// TIA Portal V17 export
// export: Created 2025-03-12T15:33:06.1888493Z, ExportSetting WithDefaults, DisplayName Totally Integrated Automation Portal, DisplayVersion V17 Update 8, DisplayName TIA Portal Openness, DisplayVersion V17 Update 8, DisplayName TIA Portal Version Control Interface, DisplayVersion V17, DisplayName SINAMICS Startdrive Advanced, DisplayVersion V17 SP2, DisplayName SINAMICS Startdrive G110M, G120, G120C, G120D, G120P, G115D, DisplayVersion V17 SP2, DisplayName SINAMICS Startdrive G130, G150, S120, S150, SINAMICS MV, S210, DisplayVersion V17 SP2, DisplayName STEP 7 Professional, DisplayVersion V17 Update 8, DisplayName SINUMERIK ONE STEP 7 Toolbox, DisplayVersion V17 Update 12, DisplayName SINUMERIK 840D sl STEP 7 Toolbox, DisplayVersion V17 Update 12, DisplayName STEP 7 Safety, DisplayVersion V17 Update 6, DisplayName WinCC Advanced, DisplayVersion V17 Update 8
FUNCTION_BLOCK "Main_Safety_RTG1"   // FB1010, F_LAD
{ S7_Optimized_Access := 'TRUE' }
VERSION : 0.1
// stored: AutoNumber false, IsIECCheckEnabled false, UDAEnableTagReadback false
   VAR
      ACK_GL_Instance : ACK_GL;
   END_VAR
BEGIN

REGION Network 1: RECEIVE SAFE I/O FROM KF900
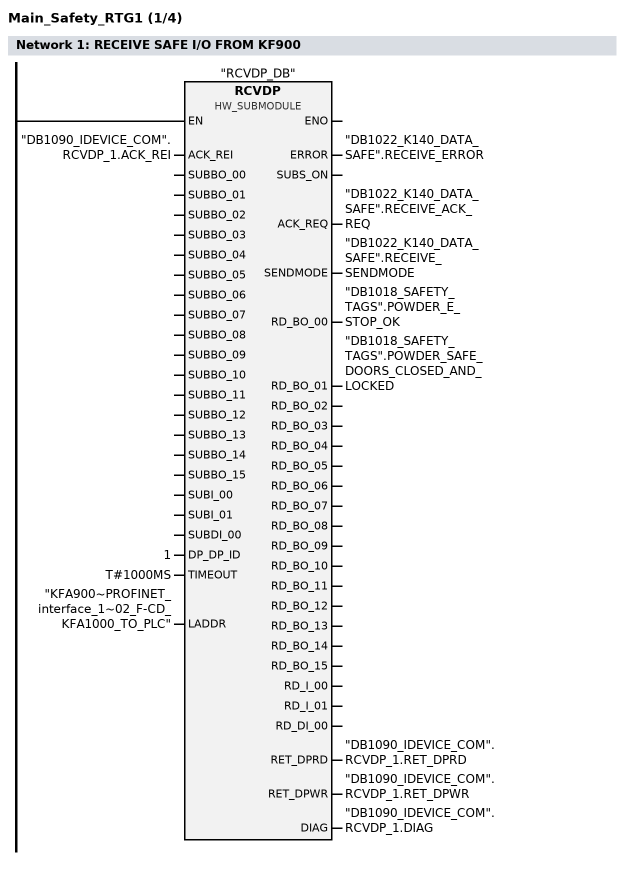
   RUNG wire#powerrail
      { S7_Templates := "laddr_type := HW_SUBMODULE" } "RCVDP_DB".RCVDP(ACK_REI := "DB1090_IDEVICE_COM".RCVDP_1.ACK_REI, SUBBO_00 :=, SUBBO_01 :=, SUBBO_02 :=, SUBBO_03 :=, SUBBO_04 :=, SUBBO_05 :=, SUBBO_06 :=, SUBBO_07 :=, SUBBO_08 :=, SUBBO_09 :=, SUBBO_10 :=, SUBBO_11 :=, SUBBO_12 :=, SUBBO_13 :=, SUBBO_14 :=, SUBBO_15 :=, SUBI_00 :=, SUBI_01 :=, SUBDI_00 :=, DP_DP_ID := 1, TIMEOUT := T#1000MS, LADDR := "KFA900~PROFINET_interface_1~02_F-CD_KFA1000_TO_PLC", ERROR => "DB1022_K140_DATA_SAFE".RECEIVE_ERROR, SUBS_ON =>, ACK_REQ => "DB1022_K140_DATA_SAFE".RECEIVE_ACK_REQ, SENDMODE => "DB1022_K140_DATA_SAFE".RECEIVE_SENDMODE, RD_BO_00 => "DB1018_SAFETY_TAGS".POWDER_E_STOP_OK, RD_BO_01 => "DB1018_SAFETY_TAGS".POWDER_SAFE_DOORS_CLOSED_AND_LOCKED, RD_BO_02 =>, RD_BO_03 =>, RD_BO_04 =>, RD_BO_05 =>, RD_BO_06 =>, RD_BO_07 =>, RD_BO_08 =>, RD_BO_09 =>, RD_BO_10 =>, RD_BO_11 =>, RD_BO_12 =>, RD_BO_13 =>, RD_BO_14 =>, RD_BO_15 =>, RD_I_00 =>, RD_I_01 =>, RD_DI_00 =>, RET_DPRD => "DB1090_IDEVICE_COM".RCVDP_1.RET_DPRD, RET_DPWR => "DB1090_IDEVICE_COM".RCVDP_1.RET_DPWR, DIAG => "DB1090_IDEVICE_COM".RCVDP_1.DIAG)
   END_RUNG
   // the same network as SCL:
   "RCVDP_DB"(ACK_REI := "DB1090_IDEVICE_COM".RCVDP_1.ACK_REI,   // RCVDP
              DP_DP_ID := 1,
              TIMEOUT := T#1000MS,
              LADDR := "KFA900~PROFINET_interface_1~02_F-CD_KFA1000_TO_PLC",
              ERROR => "DB1022_K140_DATA_SAFE".RECEIVE_ERROR,
              ACK_REQ => "DB1022_K140_DATA_SAFE".RECEIVE_ACK_REQ,
              SENDMODE => "DB1022_K140_DATA_SAFE".RECEIVE_SENDMODE,
              RD_BO_00 => "DB1018_SAFETY_TAGS".POWDER_E_STOP_OK,
              RD_BO_01 => "DB1018_SAFETY_TAGS".POWDER_SAFE_DOORS_CLOSED_AND_LOCKED,
              RET_DPRD => "DB1090_IDEVICE_COM".RCVDP_1.RET_DPRD,
              RET_DPWR => "DB1090_IDEVICE_COM".RCVDP_1.RET_DPWR,
              DIAG => "DB1090_IDEVICE_COM".RCVDP_1.DIAG);
END_REGION

REGION Network 2: RECEIVE SAFE I/O FROM ETXETAR CELL
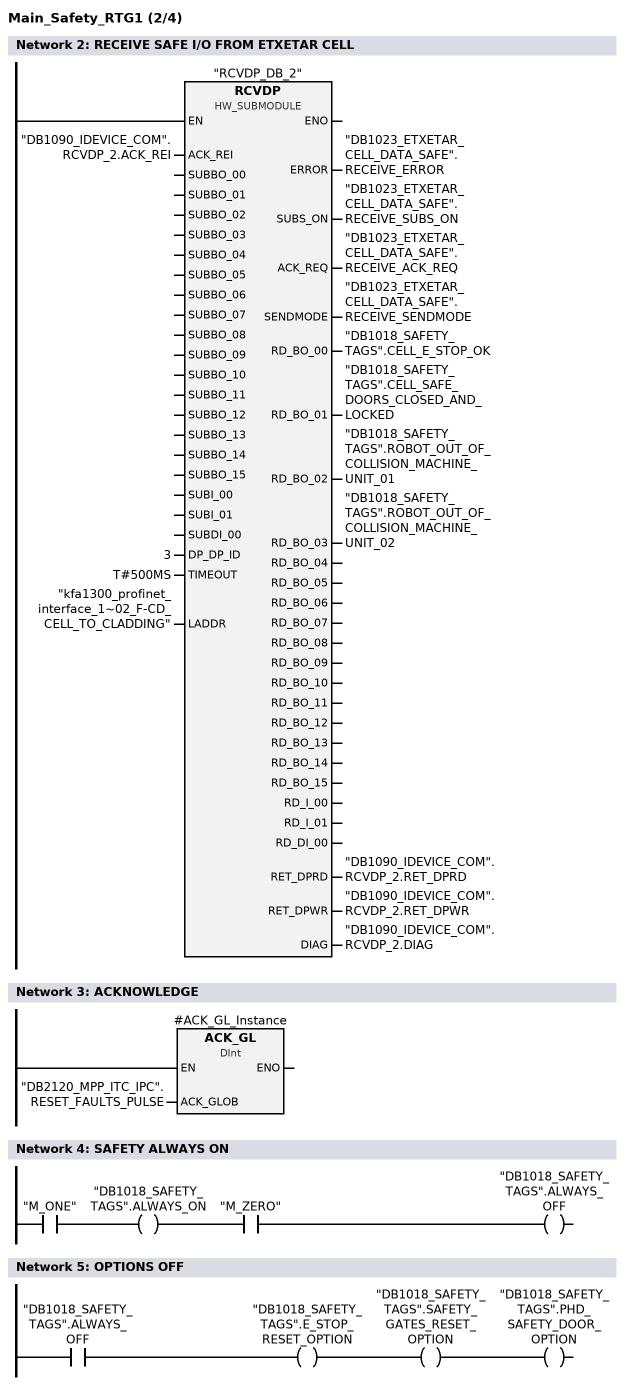
   RUNG wire#powerrail
      { S7_Templates := "laddr_type := HW_SUBMODULE" } "RCVDP_DB_2".RCVDP(ACK_REI := "DB1090_IDEVICE_COM".RCVDP_2.ACK_REI, SUBBO_00 :=, SUBBO_01 :=, SUBBO_02 :=, SUBBO_03 :=, SUBBO_04 :=, SUBBO_05 :=, SUBBO_06 :=, SUBBO_07 :=, SUBBO_08 :=, SUBBO_09 :=, SUBBO_10 :=, SUBBO_11 :=, SUBBO_12 :=, SUBBO_13 :=, SUBBO_14 :=, SUBBO_15 :=, SUBI_00 :=, SUBI_01 :=, SUBDI_00 :=, DP_DP_ID := 3, TIMEOUT := T#500MS, LADDR := "kfa1300_profinet_interface_1~02_F-CD_CELL_TO_CLADDING", ERROR => "DB1023_ETXETAR_CELL_DATA_SAFE".RECEIVE_ERROR, SUBS_ON => "DB1023_ETXETAR_CELL_DATA_SAFE".RECEIVE_SUBS_ON, ACK_REQ => "DB1023_ETXETAR_CELL_DATA_SAFE".RECEIVE_ACK_REQ, SENDMODE => "DB1023_ETXETAR_CELL_DATA_SAFE".RECEIVE_SENDMODE, RD_BO_00 => "DB1018_SAFETY_TAGS".CELL_E_STOP_OK, RD_BO_01 => "DB1018_SAFETY_TAGS".CELL_SAFE_DOORS_CLOSED_AND_LOCKED, RD_BO_02 => "DB1018_SAFETY_TAGS".ROBOT_OUT_OF_COLLISION_MACHINE_UNIT_01, RD_BO_03 => "DB1018_SAFETY_TAGS".ROBOT_OUT_OF_COLLISION_MACHINE_UNIT_02, RD_BO_04 =>, RD_BO_05 =>, RD_BO_06 =>, RD_BO_07 =>, RD_BO_08 =>, RD_BO_09 =>, RD_BO_10 =>, RD_BO_11 =>, RD_BO_12 =>, RD_BO_13 =>, RD_BO_14 =>, RD_BO_15 =>, RD_I_00 =>, RD_I_01 =>, RD_DI_00 =>, RET_DPRD => "DB1090_IDEVICE_COM".RCVDP_2.RET_DPRD, RET_DPWR => "DB1090_IDEVICE_COM".RCVDP_2.RET_DPWR, DIAG => "DB1090_IDEVICE_COM".RCVDP_2.DIAG)
   END_RUNG
   // the same network as SCL:
   "RCVDP_DB_2"(ACK_REI := "DB1090_IDEVICE_COM".RCVDP_2.ACK_REI,   // RCVDP
                DP_DP_ID := 3,
                TIMEOUT := T#500MS,
                LADDR := "kfa1300_profinet_interface_1~02_F-CD_CELL_TO_CLADDING",
                ERROR => "DB1023_ETXETAR_CELL_DATA_SAFE".RECEIVE_ERROR,
                SUBS_ON => "DB1023_ETXETAR_CELL_DATA_SAFE".RECEIVE_SUBS_ON,
                ACK_REQ => "DB1023_ETXETAR_CELL_DATA_SAFE".RECEIVE_ACK_REQ,
                SENDMODE => "DB1023_ETXETAR_CELL_DATA_SAFE".RECEIVE_SENDMODE,
                RD_BO_00 => "DB1018_SAFETY_TAGS".CELL_E_STOP_OK,
                RD_BO_01 => "DB1018_SAFETY_TAGS".CELL_SAFE_DOORS_CLOSED_AND_LOCKED,
                RD_BO_02 => "DB1018_SAFETY_TAGS".ROBOT_OUT_OF_COLLISION_MACHINE_UNIT_01,
                RD_BO_03 => "DB1018_SAFETY_TAGS".ROBOT_OUT_OF_COLLISION_MACHINE_UNIT_02,
                RET_DPRD => "DB1090_IDEVICE_COM".RCVDP_2.RET_DPRD,
                RET_DPWR => "DB1090_IDEVICE_COM".RCVDP_2.RET_DPWR,
                DIAG => "DB1090_IDEVICE_COM".RCVDP_2.DIAG);
END_REGION

REGION Network 3: ACKNOWLEDGE
   RUNG wire#powerrail
      { S7_Templates := "codedbool_type := DInt" } #ACK_GL_Instance.ACK_GL(ACK_GLOB := "DB2120_MPP_ITC_IPC".RESET_FAULTS_PULSE)
   END_RUNG
   // the same network as SCL:
   #ACK_GL_Instance(ACK_GLOB := "DB2120_MPP_ITC_IPC".RESET_FAULTS_PULSE);   // ACK_GL
END_REGION

REGION Network 4: SAFETY ALWAYS ON
   RUNG wire#powerrail
      Contact( "M_ONE" )
      Coil( "DB1018_SAFETY_TAGS".ALWAYS_ON )
      Contact( "M_ZERO" )
      Coil( "DB1018_SAFETY_TAGS".ALWAYS_OFF )
   END_RUNG
   // the same network as SCL:
   "DB1018_SAFETY_TAGS".ALWAYS_ON := "M_ONE";
   "DB1018_SAFETY_TAGS".ALWAYS_OFF := "M_ONE" AND "M_ZERO";
END_REGION

REGION Network 5: OPTIONS OFF
   RUNG wire#powerrail
      Contact( "DB1018_SAFETY_TAGS".ALWAYS_OFF )
      Coil( "DB1018_SAFETY_TAGS".E_STOP_RESET_OPTION )
      Coil( "DB1018_SAFETY_TAGS".SAFETY_GATES_RESET_OPTION )
      Coil( "DB1018_SAFETY_TAGS".PHD_SAFETY_DOOR_OPTION )
   END_RUNG
   // the same network as SCL:
   "DB1018_SAFETY_TAGS".E_STOP_RESET_OPTION := "DB1018_SAFETY_TAGS".ALWAYS_OFF;
   "DB1018_SAFETY_TAGS".SAFETY_GATES_RESET_OPTION := "DB1018_SAFETY_TAGS".ALWAYS_OFF;
   "DB1018_SAFETY_TAGS".PHD_SAFETY_DOOR_OPTION := "DB1018_SAFETY_TAGS".ALWAYS_OFF;
END_REGION

REGION Network 6: OPTIONS ON
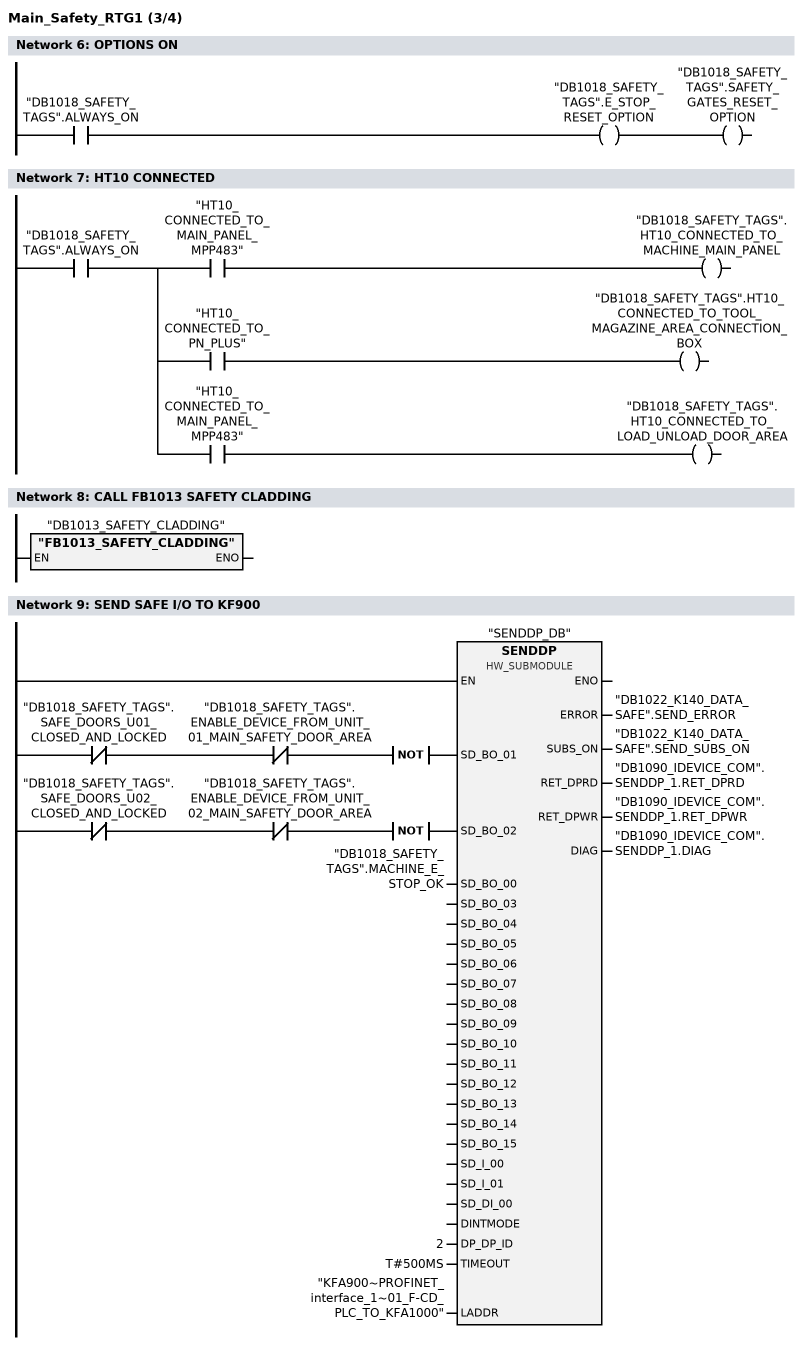
   RUNG wire#powerrail
      Contact( "DB1018_SAFETY_TAGS".ALWAYS_ON )
      Coil( "DB1018_SAFETY_TAGS".E_STOP_RESET_OPTION )
      Coil( "DB1018_SAFETY_TAGS".SAFETY_GATES_RESET_OPTION )
   END_RUNG
   // the same network as SCL:
   "DB1018_SAFETY_TAGS".E_STOP_RESET_OPTION := "DB1018_SAFETY_TAGS".ALWAYS_ON;
   "DB1018_SAFETY_TAGS".SAFETY_GATES_RESET_OPTION := "DB1018_SAFETY_TAGS".ALWAYS_ON;
END_REGION

REGION Network 7: HT10 CONNECTED
   RUNG wire#powerrail
      Contact( "DB1018_SAFETY_TAGS".ALWAYS_ON )
      wire#w1
      Contact( "HT10_CONNECTED_TO_MAIN_PANEL_MPP483" )
      Coil( "DB1018_SAFETY_TAGS".HT10_CONNECTED_TO_MACHINE_MAIN_PANEL )
   END_RUNG
   RUNG wire#w1
      Contact( "HT10_CONNECTED_TO_PN_PLUS" )
      Coil( "DB1018_SAFETY_TAGS".HT10_CONNECTED_TO_TOOL_MAGAZINE_AREA_CONNECTION_BOX )
   END_RUNG
   RUNG wire#w1
      Contact( "HT10_CONNECTED_TO_MAIN_PANEL_MPP483" )
      Coil( "DB1018_SAFETY_TAGS".HT10_CONNECTED_TO_LOAD_UNLOAD_DOOR_AREA )
   END_RUNG
   // the same network as SCL:
   "DB1018_SAFETY_TAGS".HT10_CONNECTED_TO_MACHINE_MAIN_PANEL := "DB1018_SAFETY_TAGS".ALWAYS_ON AND "HT10_CONNECTED_TO_MAIN_PANEL_MPP483";
   "DB1018_SAFETY_TAGS".HT10_CONNECTED_TO_TOOL_MAGAZINE_AREA_CONNECTION_BOX := "DB1018_SAFETY_TAGS".ALWAYS_ON AND "HT10_CONNECTED_TO_PN_PLUS";
   "DB1018_SAFETY_TAGS".HT10_CONNECTED_TO_LOAD_UNLOAD_DOOR_AREA := "DB1018_SAFETY_TAGS".ALWAYS_ON AND "HT10_CONNECTED_TO_MAIN_PANEL_MPP483";
END_REGION

REGION Network 8: CALL FB1013 SAFETY CLADDING
   RUNG wire#powerrail
      "DB1013_SAFETY_CLADDING"()
   END_RUNG
   // the same network as SCL:
   "DB1013_SAFETY_CLADDING"();   // "FB1013_SAFETY_CLADDING"
END_REGION

REGION Network 9: SEND SAFE I/O TO KF900
   RUNG wire#powerrail
      { S7_Templates := "laddr_type := HW_SUBMODULE" } "SENDDP_DB".SENDDP(SD_BO_01 := wire#w1, SD_BO_02 := wire#w2, SD_BO_00 := "DB1018_SAFETY_TAGS".MACHINE_E_STOP_OK, SD_BO_03 :=, SD_BO_04 :=, SD_BO_05 :=, SD_BO_06 :=, SD_BO_07 :=, SD_BO_08 :=, SD_BO_09 :=, SD_BO_10 :=, SD_BO_11 :=, SD_BO_12 :=, SD_BO_13 :=, SD_BO_14 :=, SD_BO_15 :=, SD_I_00 :=, SD_I_01 :=, SD_DI_00 :=, DINTMODE :=, DP_DP_ID := 2, TIMEOUT := T#500MS, LADDR := "KFA900~PROFINET_interface_1~01_F-CD_PLC_TO_KFA1000", ERROR => "DB1022_K140_DATA_SAFE".SEND_ERROR, SUBS_ON => "DB1022_K140_DATA_SAFE".SEND_SUBS_ON, RET_DPRD => "DB1090_IDEVICE_COM".SENDDP_1.RET_DPRD, RET_DPWR => "DB1090_IDEVICE_COM".SENDDP_1.RET_DPWR, DIAG => "DB1090_IDEVICE_COM".SENDDP_1.DIAG)
   END_RUNG
   RUNG wire#powerrail
      I_Contact( "DB1018_SAFETY_TAGS".SAFE_DOORS_U01_CLOSED_AND_LOCKED )
      I_Contact( "DB1018_SAFETY_TAGS".ENABLE_DEVICE_FROM_UNIT_01_MAIN_SAFETY_DOOR_AREA )
      Not()
   END_RUNG wire#w1
   RUNG wire#powerrail
      I_Contact( "DB1018_SAFETY_TAGS".SAFE_DOORS_U02_CLOSED_AND_LOCKED )
      I_Contact( "DB1018_SAFETY_TAGS".ENABLE_DEVICE_FROM_UNIT_02_MAIN_SAFETY_DOOR_AREA )
      Not()
   END_RUNG wire#w2
   // the same network as SCL:
   "SENDDP_DB"(SD_BO_01 := NOT (NOT "DB1018_SAFETY_TAGS".SAFE_DOORS_U01_CLOSED_AND_LOCKED AND NOT "DB1018_SAFETY_TAGS".ENABLE_DEVICE_FROM_UNIT_01_MAIN_SAFETY_DOOR_AREA),   // SENDDP
               SD_BO_02 := NOT (NOT "DB1018_SAFETY_TAGS".SAFE_DOORS_U02_CLOSED_AND_LOCKED AND NOT "DB1018_SAFETY_TAGS".ENABLE_DEVICE_FROM_UNIT_02_MAIN_SAFETY_DOOR_AREA),
               SD_BO_00 := "DB1018_SAFETY_TAGS".MACHINE_E_STOP_OK,
               DP_DP_ID := 2,
               TIMEOUT := T#500MS,
               LADDR := "KFA900~PROFINET_interface_1~01_F-CD_PLC_TO_KFA1000",
               ERROR => "DB1022_K140_DATA_SAFE".SEND_ERROR,
               SUBS_ON => "DB1022_K140_DATA_SAFE".SEND_SUBS_ON,
               RET_DPRD => "DB1090_IDEVICE_COM".SENDDP_1.RET_DPRD,
               RET_DPWR => "DB1090_IDEVICE_COM".SENDDP_1.RET_DPWR,
               DIAG => "DB1090_IDEVICE_COM".SENDDP_1.DIAG);
END_REGION

REGION Network 10: SEND SAFE I/O TO ETXETAR CELL
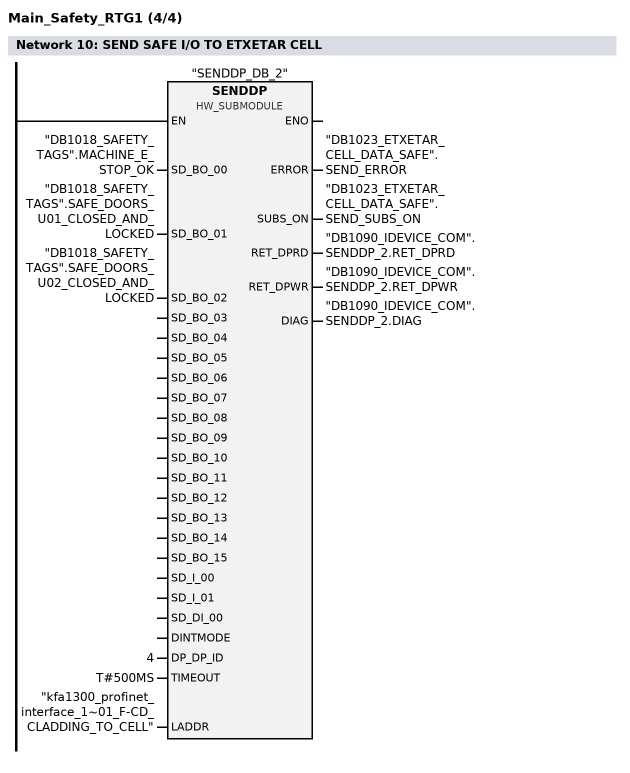
   RUNG wire#powerrail
      { S7_Templates := "laddr_type := HW_SUBMODULE" } "SENDDP_DB_2".SENDDP(SD_BO_00 := "DB1018_SAFETY_TAGS".MACHINE_E_STOP_OK, SD_BO_01 := "DB1018_SAFETY_TAGS".SAFE_DOORS_U01_CLOSED_AND_LOCKED, SD_BO_02 := "DB1018_SAFETY_TAGS".SAFE_DOORS_U02_CLOSED_AND_LOCKED, SD_BO_03 :=, SD_BO_04 :=, SD_BO_05 :=, SD_BO_06 :=, SD_BO_07 :=, SD_BO_08 :=, SD_BO_09 :=, SD_BO_10 :=, SD_BO_11 :=, SD_BO_12 :=, SD_BO_13 :=, SD_BO_14 :=, SD_BO_15 :=, SD_I_00 :=, SD_I_01 :=, SD_DI_00 :=, DINTMODE :=, DP_DP_ID := 4, TIMEOUT := T#500MS, LADDR := "kfa1300_profinet_interface_1~01_F-CD_CLADDING_TO_CELL", ERROR => "DB1023_ETXETAR_CELL_DATA_SAFE".SEND_ERROR, SUBS_ON => "DB1023_ETXETAR_CELL_DATA_SAFE".SEND_SUBS_ON, RET_DPRD => "DB1090_IDEVICE_COM".SENDDP_2.RET_DPRD, RET_DPWR => "DB1090_IDEVICE_COM".SENDDP_2.RET_DPWR, DIAG => "DB1090_IDEVICE_COM".SENDDP_2.DIAG)
   END_RUNG
   // the same network as SCL:
   "SENDDP_DB_2"(SD_BO_00 := "DB1018_SAFETY_TAGS".MACHINE_E_STOP_OK,   // SENDDP
                 SD_BO_01 := "DB1018_SAFETY_TAGS".SAFE_DOORS_U01_CLOSED_AND_LOCKED,
                 SD_BO_02 := "DB1018_SAFETY_TAGS".SAFE_DOORS_U02_CLOSED_AND_LOCKED,
                 DP_DP_ID := 4,
                 TIMEOUT := T#500MS,
                 LADDR := "kfa1300_profinet_interface_1~01_F-CD_CLADDING_TO_CELL",
                 ERROR => "DB1023_ETXETAR_CELL_DATA_SAFE".SEND_ERROR,
                 SUBS_ON => "DB1023_ETXETAR_CELL_DATA_SAFE".SEND_SUBS_ON,
                 RET_DPRD => "DB1090_IDEVICE_COM".SENDDP_2.RET_DPRD,
                 RET_DPWR => "DB1090_IDEVICE_COM".SENDDP_2.RET_DPWR,
                 DIAG => "DB1090_IDEVICE_COM".SENDDP_2.DIAG);
END_REGION
END_FUNCTION_BLOCK
